// TIA Portal V21 export
// export: Created 2026-07-07T07:59:20.9312427Z, ExportSetting WithReadOnly, DisplayName Totally Integrated Automation Portal, DisplayVersion V21, DisplayName SINAMICS Startdrive Advanced, DisplayVersion V21, DisplayName SINAMICS Startdrive G110M, G120, G120C, G120D, G120P, G115D, DisplayVersion V21, DisplayName SINAMICS Startdrive G130, G150, S120, S150, G200, G220, S200, S210, S220, Innomotics MVD, DisplayVersion V21, DisplayName STEP 7 Professional, DisplayVersion V21, DisplayName STEP 7 Safety, DisplayVersion V21, DisplayName Tech WebApplication, DisplayVersion V21, DisplayName WinCC Basic/Comfort/Advanced, DisplayVersion V21, DisplayName WinCC Professional, DisplayVersion V21, DisplayName WinCC Unified, DisplayVersion V21
DATA_BLOCK "DB1"   // DB1
{ S7_Optimized_Access := 'FALSE'; DB_Accessible_From_OPC_UA := 'FALSE' }
// stored: CodeModifiedDate 2026-07-07T07:50:54.3463936Z, CompileDate 2026-07-07T07:50:54.3509118Z, CreationDate 2026-07-07T07:50:54.2714435Z, DBAccessibleFromOPCUA false, DownloadDate 2026-07-07T07:57:30.9172103Z, InterfaceModifiedDate 2026-07-07T07:50:54.3418563Z, IsConsistent true, LoadMemoryLength 7817, ModifiedDate 2026-07-07T07:50:54.3463936Z, ParameterModified 2026-07-07T07:50:54.3418563Z, StructureModified 2026-07-07T07:50:54.3418563Z, WorkMemoryLength 304
   VAR
      EC_Set_SP : Real := 1.5;   // DBD0，SAC 输出的目标 EC
      pH_Set_SP : Real := 6.0;   // DBD4，SAC 输出的目标 pH
      EC_Actual : Real;   // DBD8，Python/传感器反馈的出口 EC
      pH_Actual : Real := 7.0;   // DBD12，Python/传感器反馈的出口 pH
      SAC_Enable : Bool;   // DBX16.0，远程/SAC 控制使能
      Reserved_17 : Byte;   // DBB17，占位，保证 Remote_Heartbeat 位于 DBW18
      Remote_Heartbeat : Int;
      Remote_Comms_OK : Bool;   // DBX20.0，PLC 判断 Python 通讯是否正常
      Reserved_21 : Byte;   // DBB21，占位，保证 Watchdog_Timer 位于 DBW22
      Watchdog_Timer : Int;
      q_f_cmd : Real;   // DBD24，PLC 输出肥料母液流量 L/min
      q_a_cmd : Real;   // DBD28，PLC 输出酸液流量 L/min
      Valve_F_Actual : Real;   // DBD32，肥液执行量反馈
      Valve_A_Actual : Real;   // DBD36，酸液执行量反馈
      AQ_Valve_F_Raw : Int;
      AQ_Valve_A_Raw : Int;
      System_Alarm_Light : Bool;   // 以下为 PLC 内部状态，不建议 Python 直接读写。
      Last_Heartbeat : Int;
      Watchdog_Count : Int;
      q_f_raw : Real;
      q_a_raw : Real;
      q_f_limited : Bool;
      q_a_limited : Bool;   // 兼容旧 A 方案/旧 OB1 网络的变量。放在 Python 固定读写区之后， 不影响 EC_Set_SP、q_f_cmd 等前 45 字节地址。
      Valve_F_Opt_SP : Real;
      Valve_A_Opt_SP : Real;
      Ramp_Target_F : Real;
      Ramp_Target_A : Real;
      Ramp_Step : Real;
      Remote_Comms_Was_OK : Bool;
      Actual_Valve_F : Real;
      Actual_Valve_A : Real;
      tWatchdog : TON_TIME;
      Growth_Stage : Int := 2;   // 0=INI, 1=DEV, 2=MID, 3=LATE
      Stage_EC_SP : Real := 1.5;   // 当前生长阶段固定 EC 保护值
      Stage_pH_SP : Real := 5.9;   // 当前生长阶段固定 pH 保护值
      Active_EC_SP : Real := 1.5;   // PLC 实际采用的 EC 目标
      Active_pH_SP : Real := 5.9;   // PLC 实际采用的 pH 目标
      Setpoint_Protection_Active : Bool;   // SAC 目标越界时置 TRUE
      Stage_Auto_SP_Enable : Bool := TRUE;   // TRUE=PLC 根据 Growth_Stage 自动写 EC_Set_SP/pH_Set_SP PID 在线调参区。Python 粗调或 TIA 监控表可直接写这些值。
      Kp_EC_Set : Real := 1.2;   // EC 比例增益
      Ki_EC_Set : Real;   // EC 积分增益
      Kd_EC_Set : Real;   // EC 微分增益
      Kp_pH_Set : Real := 1.2;   // pH 比例增益
      Ki_pH_Set : Real := 0.01;   // pH 积分增益
      Kd_pH_Set : Real;   // pH 微分增益 多肥液通道在线配置区。Enable 使用 Real(>=0.5 启用)，便于 Snap7 按 DBD 写入。
      N_Enable : Real := 1.0;   // 氮肥通道启用
      N_Ratio : Real := 0.3333;   // 总肥液 q_f_cmd 分配比例
      N_Target : Real;   // 可选氮目标；无在线 N 传感器时保持 0
      N_Actual : Real;   // 可选氮反馈；无在线 N 传感器时保持 0
      Kp_N_Set : Real;
      Ki_N_Set : Real;
      Kd_N_Set : Real;
      N_Max : Real := 4.0;
      q_n_cmd : Real;   // 氮肥计量泵输出 L/min
      AQ_Valve_N_Raw : Int;
      N_Reserved : Int;
      P_Enable : Real := 1.0;   // 磷肥通道启用
      P_Ratio : Real := 0.3333;
      P_Target : Real;
      P_Actual : Real;
      Kp_P_Set : Real;
      Ki_P_Set : Real;
      Kd_P_Set : Real;
      P_Max : Real := 4.0;
      q_p_cmd : Real;   // 磷肥计量泵输出 L/min
      AQ_Valve_P_Raw : Int;
      P_Reserved : Int;
      K_Enable : Real := 1.0;   // 钾肥通道启用
      K_Ratio : Real := 0.3334;
      K_Target : Real;
      K_Actual : Real;
      Kp_K_Set : Real;
      Ki_K_Set : Real;
      Kd_K_Set : Real;
      K_Max : Real := 4.0;
      q_k_cmd : Real;   // 钾肥计量泵输出 L/min
      AQ_Valve_K_Raw : Int;
      K_Reserved : Int;   // PLC 细调窗口：PID 只允许在前馈流量基础上做有限百分比修正。 推荐范围 0.05~0.15；0.10 表示 EC 肥液输出允许 ±10% 修正。
      EC_Trim_Band : Real := 0.1;
      pH_Trim_Band : Real := 0.08;   // 试验台本地模式区。放在现有 Python 固定地址区之后，避免改变既有 offset。
      Manual_Mode : Bool;   // TRUE=手动调试模式，绕过 EC/pH 自动闭环
      Auto_Mode : Bool;   // TRUE=预留本地自动模式，当前自动仍由 SAC_Enable 驱动
      Emergency_Stop : Bool;   // TRUE=急停，所有执行量立即归零
      Manual_Active : Bool;   // PLC 当前处于手动输出
      Auto_Active : Bool;   // PLC 当前处于自动闭环输出
      Reserved_279 : Byte;   // 占位，使 Manual_q_* 从 DBD280 开始
      Manual_q_f_Set : Real;   // 手动总肥液流量 L/min，限幅 0~10
      Manual_q_a_Set : Real;   // 手动酸液流量 L/min，限幅 0~4
      Manual_q_n_Set : Real;   // 手动氮肥通道 L/min，限幅 0~N_Max
      Manual_q_p_Set : Real;   // 手动磷肥通道 L/min，限幅 0~P_Max
      Manual_q_k_Set : Real;   // 手动钾肥通道 L/min，限幅 0~K_Max
   END_VAR
BEGIN
END_DATA_BLOCK
